// TIA Portal project "Project_PNPNCoupler" (V15.1)

(* hardware
DEVICE "S7-1200 station_1"  S7-1200 Station
   slot 0: "Rack_0"  S7-1200 Rack  Rack  V1.0
   slot 1: "PLC_1"  CPU 1212FC DC/DC/DC  6ES7 212-1AF40-0XB0  V4.2
DEVICE "GSD device_1"  GSD.Device.PN
   slot 0: "Rack"  Rack  V1.0
   slot 0: "PNPN-CouplerX1"  PN/PN Coupler X1  6ES7 158-3AD10-0XA0  V04.02.00
      slot 0: "PN/PN Coupler X1"  PN/PN Coupler X1
      slot 1: "PN-IO-01"  PN-IO-01
   slot 1: "Port 1 (2xRJ45)"  Port 1 (2xRJ45)  6ES7 193-6AR00-0AA0
   slot 1: "IN 253 Byte+DS_1"  IN 253 Byte+DS
      slot 0: "IN 253 Byte+DS"  IN 253 Byte+DS
   slot 2: "Port 2 (2xRJ45)"  Port 2 (2xRJ45)  6ES7 193-6AR00-0AA0
   slot 2: "OUT 253 Byte_1"  OUT 253 Byte
      slot 0: "OUT 253 Byte"  OUT 253 Byte
*)

// ===== PLC "PLC_1"  CPU 1212FC DC/DC/DC =====

VAR_GLOBAL   // PLC tag table "Default tag table"
   "Tag_1" AT %MW2 : Int;
   "Tag_2" AT %MW4 : Int;
END_VAR

DATA_BLOCK "dbGet"   // DB1
{ S7_Optimized_Access := 'FALSE' }
VERSION : 0.1
   VAR
      UDINT : Array[0..62] of UDInt;
      USINT : USInt;
      DS : USInt;
   END_VAR
BEGIN
END_DATA_BLOCK

DATA_BLOCK "dbPut"   // DB2
{ S7_Optimized_Access := 'FALSE' }
VERSION : 0.1
   VAR
      UDINT : Array[0..62] of UDInt;
      "BYTE" : Byte;
   END_VAR
BEGIN
END_DATA_BLOCK

ORGANIZATION_BLOCK "Main"   // OB1, LAD, ProgramCycle
TITLE = "Main Program Sweep (Cycle)"
{ S7_Optimized_Access := 'TRUE' }
VERSION : 0.1
   VAR_INPUT
      Initial_Call : Bool;   // Initial call of this OB
      Remanence : Bool;   // =True, if remanent data are available
   END_VAR
BEGIN

REGION Network 2
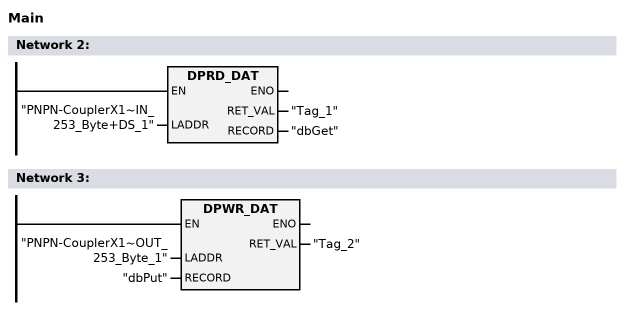
   "Tag_1" := DPRD_DAT(LADDR := "PNPN-CouplerX1~IN_253_Byte+DS_1", RECORD => "dbGet");
END_REGION

REGION Network 3
   "Tag_2" := DPWR_DAT(LADDR := "PNPN-CouplerX1~OUT_253_Byte_1", RECORD := "dbPut");
END_REGION
END_ORGANIZATION_BLOCK

ORGANIZATION_BLOCK "Diagnostic error interrupt"   // OB82, LAD, DiagnosticErrorInterrupt
{ S7_Optimized_Access := 'TRUE' }
VERSION : 0.1
   VAR_INPUT
      IO_State : Word;   // IO state of the HW object
      LADDR : Hw_Any;   // Hardware identifier
      Channel : UInt;   // Channel number
      MultiError : Bool;   // =true if more than one error is present
   END_VAR
BEGIN
END_ORGANIZATION_BLOCK

ORGANIZATION_BLOCK "Pull or plug of modules"   // OB83, LAD, PullPlug
{ S7_Optimized_Access := 'TRUE' }
VERSION : 0.1
   VAR_INPUT
      LADDR : Hw_Io;   // Hardware identifier
      Event_Class : Byte;   // 16#38/39: module inserted, removed
      Fault_ID : Byte;   // Fault identifier
   END_VAR
BEGIN
END_ORGANIZATION_BLOCK

ORGANIZATION_BLOCK "Rack or station failure"   // OB86, LAD, RackStationFailure
{ S7_Optimized_Access := 'TRUE' }
VERSION : 0.1
   VAR_INPUT
      LADDR : Hw_Device;   // Hardware identifier
      Event_Class : Byte;   // Event class
      Fault_ID : Byte;   // Fault identifier
   END_VAR
BEGIN
END_ORGANIZATION_BLOCK